(* IEC 61131-3 sources: volt/packages/volt-lsp-iec/test-corpus/pro2193/Device/Plc Logic/Application/99 Library/Function Blocks/Actuators/Cylinders, 8 files *)

(* ---- Cylinder_52Valve_InvertedFB.pou ---- *)
// Control a single output (e.g. a cylinder). Two sensors check if the cylinder is in position. The output is inverted
{attribute 'monitoring_display' := 'Output.output'}
{attribute 'symbol' := 'none'}
FUNCTION_BLOCK PUBLIC Cylinder_52Valve_InvertedFB
EXTENDS Cylinder_52ValveFB
IMPLEMENTS IActuator

%LANGUAGE ST
// Execute base cylinder fb
SUPER^();

END_FUNCTION_BLOCK

METHOD PROTECTED Alarms

%LANGUAGE ST
// Set the alarm messages (inverted)
SetSensorOutAlarm(	inputIn XOR NOT Output.Map());
SetSensorInAlarm(	inputOut XOR Output.Map());

END_METHOD

// The cylinder moves in. Returns true when cylinder is in. (Inverted!)
METHOD PUBLIC FINAL GoIn : BOOL

%LANGUAGE ST
SUPER^.GoOut();

GoIn := IsIn;

END_METHOD

// The cylinder moves out. Returns true when cylinder is out. (Inverted!)
METHOD PUBLIC FINAL GoOut : BOOL

%LANGUAGE ST
SUPER^.GoIn();

GoOut := IsOut;

END_METHOD

// Reset the output (=True, because inverted!)
METHOD Reset

%LANGUAGE ST
SUPER^.Set();

END_METHOD

// Set the output (=False, because inverted!)
METHOD Set

%LANGUAGE ST
SUPER^.Reset();

END_METHOD

// Set the output True or False (Inverted!)
METHOD SetOrReset
VAR_INPUT
	xValue	: BOOL;
END_VAR

%LANGUAGE ST
SUPER^.SetOrReset(NOT xValue);

END_METHOD

{attribute 'monitoring':='call'}
PROPERTY IsIn : BOOL

GET
VAR
END_VAR

%LANGUAGE ST
IsIn := SUPER^.IsOut;
END_GET
END_PROPERTY

{attribute 'monitoring':='call'}
PROPERTY IsOut : BOOL

GET
VAR
END_VAR

%LANGUAGE ST
IsOut := SUPER^.IsIn;
END_GET
END_PROPERTY

(* ---- Cylinder_52Valve_TimedFB.pou ---- *)
// Control a single output (e.g. a cylinder). No sensors, use timers to check cylinder position. Sensor inputs are ignored. Alarms are disabled.
{attribute 'monitoring_display' := 'Output.output'}
{attribute 'symbol' := 'none'}
FUNCTION_BLOCK PUBLIC Cylinder_52Valve_TimedFB
EXTENDS ActuatorWithManualControl_BaseFB
IMPLEMENTS IActuator
VAR_INPUT
	rTimeToGoIn				: REAL	:= 0.3;		// Time it should take for the cylinder to move in.
	rTimeToGoOut			: REAL	:= 0.3;		// Time it should take for the cylinder to move out.
END_VAR
VAR
	{attribute 'symbol' := 'read'}		Output					: ActuatorFB;

	timeGoOut				: BTON;
	timeGoIn				: BTON;

	{attribute 'symbol' := 'readwrite'}	adjustButton			: BOOL;		// Enable adjust mode for cylinder
	adjustTrigger			: TriggerFB;
	{attribute 'hide'}
	Blinker					: BLINK;	// Blinker for adjust mode
	inAdjustMode			: BOOL;		// When high the cylinder moves automatically
	SetAdjustModeTimer		: BTON;

END_VAR
VAR CONSTANT
	tAdjustFrequency		: TIME	:= T#2S;
END_VAR

%LANGUAGE ST
// Execute base fb
SUPER^();

// Instantiate the output
Output();

timeGoIn.Set(	In := NOT Output.Map(),	Pt := rTimeToGoIn);
timeGoOut.Set(	In := Output.Map(),		Pt := rTimeToGoOut);

IF adjustTrigger.Rising(CLK := adjustButton) THEN
	inAdjustMode := NOT inAdjustMode;
END_IF

inAdjustMode	S= SetAdjustModeTimer.Set(In := hardwareF1Pushed AND hardwareF2Pushed, Pt := 5);
inAdjustMode	R= plusTrigger.Q_Rising;
inAdjustMode	R= minTrigger.Q_Rising;

GlobalVars.manualControlRequested S= inAdjustMode;

Blinker(ENABLE := inAdjustMode, TIMELOW := tAdjustFrequency, TIMEHIGH := tAdjustFrequency);

END_FUNCTION_BLOCK

// The cylinder moves in. Returns true when cylinder is in.
METHOD PUBLIC FINAL GoIn : BOOL

%LANGUAGE ST
Reset();

GoIn := IsIn;

END_METHOD

// The cylinder moves out. Returns true when cylinder is out.
METHOD PUBLIC FINAL GoOut : BOOL

%LANGUAGE ST
Set();

GoOut := IsOut;

END_METHOD

METHOD PROTECTED ManualControl
VAR_INPUT
	minButtonPushed			: BOOL;		// Both the software button (on screen) and the hardware button (if attached)
	plusButtonPushed		: BOOL;		// Both the software button (on screen) and the hardware button (if attached)
END_VAR

%LANGUAGE ST
IF inAdjustMode THEN
	SetOrReset(Blinker.OUT);
ELSIF plusButtonPushed THEN
	GoOut();
ELSIF minButtonPushed THEN
	GoIn();
END_IF

END_METHOD

// Maps the actuator to the physical output
METHOD Map : BOOL

%LANGUAGE ST
Map := Output.Map();

END_METHOD

// Reset the output (=False)
METHOD Reset

%LANGUAGE ST
Output.Reset();

END_METHOD

// Set the output (=True)
METHOD Set : BOOL

%LANGUAGE ST
Output.Set();

END_METHOD

// Set the output True or False
METHOD SetOrReset
VAR_INPUT
	xValue	: BOOL;
END_VAR

%LANGUAGE ST
Output.SetOrReset(xValue);

END_METHOD

{attribute 'monitoring':='call'}
PROPERTY IsIn : BOOL

GET
VAR
END_VAR

%LANGUAGE ST
IsIn := timeGoIn.Q;
END_GET
END_PROPERTY

{attribute 'monitoring':='call'}
PROPERTY IsOut : BOOL

GET
VAR
END_VAR

%LANGUAGE ST
IsOut := timeGoOut.Q;
END_GET
END_PROPERTY

(* ---- Cylinder_52ValveFB.pou ---- *)
// Control a single output (e.g. a cylinder). Two sensors check if the cylinder is in position.
{attribute 'monitoring_display' := 'Output.output'}
{attribute 'symbol' := 'none'}
FUNCTION_BLOCK PUBLIC Cylinder_52ValveFB
EXTENDS Cylinder_BaseFB
IMPLEMENTS IActuator
VAR
	{attribute 'symbol' := 'read'}	Output					: ActuatorFB;
END_VAR

%LANGUAGE ST
// Execute base cylinder fb
SUPER^();

// Instantiate the output
Output();

END_FUNCTION_BLOCK

METHOD PROTECTED Alarms

%LANGUAGE ST
// Set the alarm messages
SetSensorOutAlarm(	inputOut XOR Output.Map());
SetSensorInAlarm(	inputIn XOR NOT Output.Map());

END_METHOD

// The cylinder moves in. Returns true when cylinder is in.
METHOD PUBLIC FINAL GoIn : BOOL

%LANGUAGE ST
Reset();

GoIn := IsIn;

END_METHOD

// The cylinder moves out. Returns true when cylinder is out.
METHOD PUBLIC FINAL GoOut : BOOL

%LANGUAGE ST
Set();

GoOut := IsOut;

END_METHOD

METHOD PROTECTED ManualControl
VAR_INPUT
	minButtonPushed			: BOOL;		// Both the software button (on screen) and the hardware button (if attached)
	plusButtonPushed		: BOOL;		// Both the software button (on screen) and the hardware button (if attached)
END_VAR

%LANGUAGE ST
IF inAdjustMode THEN
	SetOrReset(Blinker.OUT);
ELSIF plusButtonPushed THEN
	GoOut();
ELSIF minButtonPushed THEN
	GoIn();
END_IF

END_METHOD

// Maps the actuator to the physical output
METHOD Map : BOOL

%LANGUAGE ST
Map := Output.Map();

END_METHOD

// Reset the output (=False)
METHOD Reset

%LANGUAGE ST
Output.Reset();

END_METHOD

// Set the output (=True)
METHOD Set : BOOL

%LANGUAGE ST
Output.Set();

END_METHOD

// Set the output True or False
METHOD SetOrReset
VAR_INPUT
	xValue	: BOOL;
END_VAR

%LANGUAGE ST
Output.SetOrReset(xValue);

END_METHOD

(* ---- Cylinder_53Valve_InvertedFB.pou ---- *)
// Control a dual output cylinder. Two sensors check if the cylinder is in position. The outputs are inverted
{attribute 'symbol' := 'none'}
FUNCTION_BLOCK FINAL Cylinder_53Valve_InvertedFB
EXTENDS Cylinder_53ValveFB
IMPLEMENTS IActuator

%LANGUAGE ST
// Execute base cylinder fb
SUPER^();

END_FUNCTION_BLOCK

METHOD PROTECTED Alarms

%LANGUAGE ST
// Set the alarm messages (inverted)
SetSensorOutAlarm(	SetAlarm(OutputOut.Map(), OutputIn.Map(), inputIn));
SetSensorInAlarm(	SetAlarm(OutputIn.Map(), OutputOut.Map(), inputOut));

END_METHOD

// The cylinder moves in. Returns true when cylinder is in. (Inverted!)
METHOD PUBLIC GoIn : BOOL

%LANGUAGE ST
SUPER^.GoOut();

GoIn := IsIn;

END_METHOD

// The cylinder moves out. Returns true when cylinder is out. (Inverted!)
METHOD PUBLIC GoOut : BOOL

%LANGUAGE ST
SUPER^.GoIn();

GoOut := IsOut;

END_METHOD

// Set the output True or False (Inverted!)
METHOD SetOrReset
VAR_INPUT
	xValue	: BOOL;
END_VAR

%LANGUAGE ST
SUPER^.SetOrReset(NOT xValue);

END_METHOD

{attribute 'monitoring':='call'}
PROPERTY IsIn : BOOL

GET
VAR
END_VAR

%LANGUAGE ST
IsIn := SUPER^.IsOut;

END_GET
END_PROPERTY

{attribute 'monitoring':='call'}
PROPERTY IsOut : BOOL

GET
VAR
END_VAR

%LANGUAGE ST
IsOut := SUPER^.IsIn;
END_GET
END_PROPERTY

{attribute 'monitoring':='call'}
PROPERTY OnTargetPos : BOOL

GET
VAR
END_VAR

%LANGUAGE ST
OnTargetPos	:= NOT SUPER^.OnTargetPos;
END_GET
END_PROPERTY

(* ---- Cylinder_53Valve_InvertibleFB.pou ---- *)
// Control a dual output cylinder. Two sensors check if the cylinder is in position. The outputs can be inverted
{attribute 'symbol' := 'none'}
FUNCTION_BLOCK FINAL Cylinder_53Valve_InvertibleFB
EXTENDS Cylinder_53ValveFB
IMPLEMENTS IActuator
VAR_INPUT
	xInvertOutput			: BOOL;
END_VAR

%LANGUAGE ST
// Execute base cylinder fb
SUPER^();

END_FUNCTION_BLOCK

METHOD PROTECTED Alarms

%LANGUAGE ST
// Set the alarm messages (inverted)
IF xInvertOutput THEN
	SetSensorOutAlarm(	SetAlarm(OutputOut.Map(), OutputIn.Map(), inputIn));
	SetSensorInAlarm(	SetAlarm(OutputIn.Map(), OutputOut.Map(), inputOut));
ELSE
	SUPER^.Alarms();
END_IF

END_METHOD

// The cylinder moves in. Returns true when cylinder is in. (Optionally inverted!)
METHOD PUBLIC GoIn : BOOL

%LANGUAGE ST
IF xInvertOutput THEN
	SUPER^.GoOut();
ELSE
	SUPER^.GoIn();
END_IF

GoIn := IsIn;

END_METHOD

// The cylinder moves out. Returns true when cylinder is out. (Optionally inverted!)
METHOD PUBLIC GoOut : BOOL

%LANGUAGE ST
IF xInvertOutput THEN
	SUPER^.GoIn();
ELSE
	SUPER^.GoOut();
END_IF

GoOut := IsOut;

END_METHOD

// Set the output True or False
METHOD SetOrReset
VAR_INPUT
	xValue	: BOOL;
END_VAR

%LANGUAGE ST
IF xInvertOutput THEN
	SUPER^.SetOrReset(NOT xValue);
ELSE
	SUPER^.SetOrReset(xValue);
END_IF

END_METHOD

{attribute 'monitoring':='call'}
PROPERTY IsIn : BOOL

GET
VAR
END_VAR

%LANGUAGE ST
IF xInvertOutput THEN
	IsIn := SUPER^.IsOut;
ELSE
	IsIn := SUPER^.IsIn;
END_IF

END_GET
END_PROPERTY

{attribute 'monitoring':='call'}
PROPERTY IsOut : BOOL

GET
VAR
END_VAR

%LANGUAGE ST
IF xInvertOutput THEN
	IsOut := SUPER^.IsIn;
ELSE
	IsOut := SUPER^.IsOut;
END_IF

END_GET
END_PROPERTY

{attribute 'monitoring':='call'}
PROPERTY OnTargetPos : BOOL

GET
VAR
END_VAR

%LANGUAGE ST
IF xInvertOutput THEN
	OnTargetPos := NOT SUPER^.OnTargetPos;
ELSE
	OnTargetPos := SUPER^.OnTargetPos;
END_IF

END_GET
END_PROPERTY

(* ---- Cylinder_53Valve_MiddleSensorFB.pou ---- *)
// Control a dual output cylinder. Three sensors check if the cylinder is in position. Middle sensor is high when both outputs are turned off.
{attribute 'symbol' := 'none'}
FUNCTION_BLOCK FINAL Cylinder_53Valve_MiddleSensorFB
EXTENDS Cylinder_53ValveFB
VAR_INPUT
	{attribute 'symbol' := 'read'}	xSensorMiddle			: BOOL;
	errorId_SensorMiddle	: WORD;
END_VAR
VAR
	SensorMiddleAlarm		: SetErrorFB;
	{attribute 'symbol' := 'read'}		moveMiddleDuration		: REAL;		// The amount of time elapsed when cylinder moves
END_VAR

%LANGUAGE ST
// Execute base cylinder fb
SUPER^();

END_FUNCTION_BLOCK

METHOD PROTECTED Alarms

%LANGUAGE ST
// Set the extra alarm message
SUPER^.Alarms();
SetSensorMiddleAlarm(	(OutputIn.Map() = OutputOut.Map()) XOR xSensorMiddle);

END_METHOD

METHOD PROTECTED SetSensorMiddleAlarm
VAR_INPUT
	xSet	: BOOL;
END_VAR

%LANGUAGE ST
SensorMiddleAlarm(
	moduleHandler	:= moduleHandler,
	textRefId		:= textRefId,
	alarmCondition	:= alarmEnable AND xSet AND errorId_SensorMiddle <> 0,
	alarmDelay		:= alarmDelay,
	errorId			:= errorId_SensorMiddle,
	severity		:= severity,
	reaction		:= reaction,
	active			=> );

IF alarmEnable AND xSet AND errorId_SensorIn <> 0 THEN
	moveMiddleDuration	:= SensorMiddleAlarm.ElapsedTime;
END_IF

END_METHOD

{attribute 'monitoring':='call'}
PROPERTY IsIn : BOOL

GET
VAR
END_VAR

%LANGUAGE ST
IsIn := inputIn AND NOT inputOut AND NOT xSensorMiddle;
END_GET
END_PROPERTY

{attribute 'monitoring':='call'}
PROPERTY IsMiddle : BOOL

GET
VAR
END_VAR

%LANGUAGE ST
IsMiddle := NOT inputOut AND NOT inputIn AND xSensorMiddle;
END_GET
END_PROPERTY

{attribute 'monitoring':='call'}
PROPERTY IsOut : BOOL

GET
VAR
END_VAR

%LANGUAGE ST
IsOut := inputOut AND NOT inputIn AND NOT xSensorMiddle;
END_GET
END_PROPERTY

(* ---- Cylinder_53ValveFB.pou ---- *)
// Control a dual output cylinder. Two sensors check if the cylinder is in position.
{attribute 'symbol' := 'none'}
FUNCTION_BLOCK PUBLIC Cylinder_53ValveFB
EXTENDS Cylinder_BaseFB
IMPLEMENTS IActuator
VAR_INPUT
	rGiveAirToBothOutputs	: REAL := 0.2;	// When a 5/3 valve is set while both outputs are low, give air to both outputs for this time. To avoid fast moving cylinder. Default is 200MS.
	xEnableOutputs			: BOOL;			// Use like this: 'G_xEnableMainvalve OR System.On'. Resets outputs when air pressure is killed. Alarms are disables when low. Set to TRUE to disable this feature.
END_VAR
VAR
	{attribute 'symbol' := 'readwrite'}	middleButton			: BOOL;			// Enable adjust mode for cylinder
	{attribute 'symbol' := 'read'}		OutputIn				: ActuatorFB;	// Output when cylinder moves in
	{attribute 'symbol' := 'read'}		OutputOut				: ActuatorFB;	// Output when cylinder moves out

	middleTrigger			: TriggerFB;

	switchBothOutputs		: BTON;
	EnableOutputs			: BTOF;
	xStartGoInDelay			: BOOL;
	xStartGoOutDelay		: BOOL;
END_VAR

%LANGUAGE ST
// Execute base cylinder fb
SUPER^();

// Instantiate the outputs
OutputIn();
OutputOut();

// Keep xEnableOutputs high for half a second. So if air pressure drops for 0,5 sec. the outputs are reset.
IF NOT EnableOutputs.Set(In := xEnableOutputs, Pt := 0.5) THEN
	Reset();
END_IF

switchBothOutputs.Set(
	In := xStartGoInDelay OR xStartGoOutDelay,
	Pt := rGiveAirToBothOutputs);

IF switchBothOutputs.Q THEN
	SetOrReset(xStartGoOutDelay);
	xStartGoInDelay		:= FALSE;
	xStartGoOutDelay	:= FALSE;
END_IF

IF middleButton THEN
	GlobalVars.manualControlRequested := TRUE;
END_IF

END_FUNCTION_BLOCK

METHOD PROTECTED Alarms

%LANGUAGE ST
// Set the alarm messages
SetSensorOutAlarm(
	SetAlarm(
		xOutput	:= OutputOut.Map(),
		xOutInv	:= OutputIn.Map(),
		xSensor	:= inputOut));

SetSensorInAlarm(
	SetAlarm(
		xOutput	:= OutputIn.Map(),
		xOutInv	:= OutputOut.Map(),
		xSensor	:= inputIn));

END_METHOD

// Set both outputs (=True)
METHOD PUBLIC FINAL GoForceMiddle : BOOL

%LANGUAGE ST
OutputIn.Set();
OutputOut.Set();

END_METHOD

// The cylinder moves in. Returns true when cylinder is in.
METHOD PUBLIC GoIn : BOOL

%LANGUAGE ST
// Do not move cylinder if outputs are not enabled.
IF NOT EnableOutputs.Q THEN
	RETURN;
END_IF

// Both outputs are switched off, and the cylinder is not already in position
IF NOT OutputIn.Map() AND NOT OutputOut.Map() AND NOT inputIn THEN
	IF inputOut THEN		// Cylinder is on the opposite side
		OutputOut.Set();		// Send cylinder to opposite direction
		OutputIn.Reset();
		xStartGoInDelay	:= TRUE;
	ELSE					// Cylinder is in between sensors
		GoForceMiddle();	// Give air to both sides of the cylinder
		xStartGoInDelay	:= TRUE;
	END_IF
ELSIF NOT xStartGoInDelay THEN
	OutputOut.Reset();
	OutputIn.Set();

	GoIn := IsIn;
END_IF

END_METHOD

// Reset both outputs. The 5/3 valve goes to middle position.
METHOD PUBLIC GoMiddle

%LANGUAGE ST
Reset();
END_METHOD

// The cylinder moves out. Returns true when cylinder is out.
METHOD PUBLIC GoOut : BOOL

%LANGUAGE ST
// Do not move cylinder if outputs are not enabled.
IF NOT EnableOutputs.Q THEN
	RETURN;
END_IF

// Both outputs are switched off, and the cylinder is not already in position
IF NOT OutputIn.Map() AND NOT OutputOut.Map() AND NOT inputOut THEN
	IF inputIn THEN		// Cylinder is on the opposite side
		OutputOut.Reset();
		OutputIn.Set();		// Send cylinder to opposite direction
		xStartGoOutDelay	:= TRUE;
	ELSE					// Cylinder is in between sensors
		GoForceMiddle();	// Give air to both sides of the cylinder
		xStartGoOutDelay	:= TRUE;
	END_IF
ELSIF NOT xStartGoOutDelay THEN
	OutputOut.Set();
	OutputIn.Reset();

	GoOut := IsOut;
END_IF

END_METHOD

METHOD PROTECTED ManualControl
VAR_INPUT
	minButtonPushed			: BOOL;		// Both the software button (on screen) and the hardware button (if attached)
	plusButtonPushed		: BOOL;		// Both the software button (on screen) and the hardware button (if attached)
END_VAR

%LANGUAGE ST
IF inAdjustMode THEN
	SetOrReset(Blinker.OUT);
ELSIF plusButtonPushed THEN
	IF OutputOut.Map() THEN
		GoMiddle();
	ELSE
		GoOut();
	END_IF
ELSIF minButtonPushed THEN
	IF OutputIn.Map() THEN
		GoMiddle();
	ELSE
		GoIn();
	END_IF
ELSIF middleTrigger.Rising(CLK := middleButton) THEN
	GoMiddle();
END_IF

END_METHOD

{attribute 'hide'}
METHOD Map : BOOL

%LANGUAGE ST
ThrowException('Use other mapping methods instead');

END_METHOD

// Maps the output when cylinder moves Out to the physical output
METHOD MapIn : BOOL

%LANGUAGE ST
MapIn := OutputIn.Map();

END_METHOD

// Maps the output when cylinder moves Out to the physical output
METHOD MapOut : BOOL

%LANGUAGE ST
MapOut := OutputOut.Map();

END_METHOD

// Reset the outputs (=False)
METHOD Reset

%LANGUAGE ST
OutputIn.Reset();
OutputOut.Reset();

END_METHOD

// Set the outputs (=True)
METHOD Set : BOOL

%LANGUAGE ST
GoOut();

END_METHOD

METHOD PRIVATE SetAlarm : BOOL
VAR_INPUT
	xOutput		: BOOL;		// The output
	xOutInv		: BOOL;		// The output that moves the cylinder the other way.
	xSensor		: BOOL;		// The sensor on the cylinder.
END_VAR

%LANGUAGE FBD
%NETWORK
ASSIGN(AND(AND(xOutput, INVERT(xOutInv), INVERT(xSensor)) OR AND(xOutInv, INVERT(xOutput), xSensor) OR AND(xOutput, xOutInv, xSensor), EnableOutputs.Q), Q => SetAlarm);
END_METHOD

// Set the output True or False
METHOD SetOrReset
VAR_INPUT
	xValue	: BOOL;
END_VAR

%LANGUAGE ST
// Do not move cylinder if outputs are not enabled.
IF NOT EnableOutputs.Q THEN
	RETURN;
END_IF

// Timer expired, so both outputs are high. Just switch to desired output.
IF switchBothOutputs.Q THEN
	OutputOut.SetOrReset(xValue);
	OutputIn.SetOrReset(NOT xValue);
// Both outputs are switched off. Give air to both sides of the valve. Start timer.
ELSIF NOT OutputIn.Map() AND NOT OutputOut.Map() THEN
	GoForceMiddle();
	xStartGoInDelay		:= NOT xValue;	// Choose direction to move to when timer expires.
	xStartGoOutDelay	:= xValue;
// Normal operation
ELSIF NOT xStartGoInDelay AND NOT xStartGoOutDelay THEN
	OutputOut.SetOrReset(xValue);
	OutputIn.SetOrReset(NOT xValue);
END_IF

END_METHOD

// Set both the outputs of the valve immediately
METHOD SetOrResetBothOutputs : BOOL
VAR_INPUT
	xOutput2	: BOOL;		// Output when cylinder moves out
	xOutput1	: BOOL;		// Output when cylinder moves in
END_VAR

%LANGUAGE ST
OutputOut.SetOrReset(xOutput2);
OutputIn.SetOrReset(xOutput1);

END_METHOD

{attribute 'monitoring':='call'}
PROPERTY OnTargetPos : BOOL

GET
VAR
END_VAR

%LANGUAGE ST
OnTargetPos	:= NOT xStartGoInDelay AND NOT xStartGoOutDelay AND EnableOutputs.Q AND
			(OutputOut.Map() AND NOT OutputIn.Map() AND IsOut) XOR (OutputIn.Map() AND NOT OutputOut.Map() AND IsIn);

END_GET
END_PROPERTY

(* ---- Cylinder_BaseFB.pou ---- *)
// Abstract Base fb for cylinders. Has general stuff for all cylinder types.
{attribute 'symbol' := 'none'}
FUNCTION_BLOCK PUBLIC ABSTRACT Cylinder_BaseFB
EXTENDS ActuatorWithManualControlAndAlarm_BaseFB
VAR_INPUT
	{attribute 'symbol' := 'read'}		inputOut				: BOOL;
	{attribute 'symbol' := 'read'}		inputIn					: BOOL;
	errorId_SensorOut		: WORD;		// Set to ZERO if OUT sensor is not on the cylinder, this will prevent incorrect alarm messages.
	errorId_SensorIn		: WORD;		// Set to ZERO if IN sensor is not on the cylinder, this will prevent incorrect alarm messages.
END_VAR
VAR
	SensorOutAlarm			: SetErrorFB;
	SensorInAlarm			: SetErrorFB;
	{attribute 'symbol' := 'read'}		moveInDuration			: REAL;		// The amount of time elapsed when cylinder moves out
	{attribute 'symbol' := 'read'}		moveOutDuration			: REAL;		// The amount of time elapsed when cylinder moves in

	MeasureMaxTimeIn		: StopwatchFB;
	MeasureMaxTimeOut		: StopwatchFB;

	{attribute 'symbol' := 'readwrite'}	adjustButton			: BOOL;		// Enable adjust mode for cylinder
	adjustTrigger			: TriggerFB;
	{attribute 'hide'}
	Blinker					: BLINK;	// Blinker for adjust mode
	inAdjustMode			: BOOL;		// When high the cylinder moves automatically
	SetAdjustModeTimer		: BTON;
END_VAR
VAR CONSTANT
	tAdjustFrequency		: TIME	:= T#2S;
END_VAR

%LANGUAGE ST
SUPER^();

IF adjustTrigger.Rising(CLK := adjustButton) THEN
	inAdjustMode := NOT inAdjustMode;
END_IF

inAdjustMode	S= SetAdjustModeTimer.Set(In := hardwareF1Pushed AND hardwareF2Pushed, Pt := 5);
inAdjustMode	R= plusTrigger.Q_Rising;
inAdjustMode	R= minTrigger.Q_Rising;

GlobalVars.manualControlRequested S= inAdjustMode;

Blinker(ENABLE := inAdjustMode, TIMELOW := tAdjustFrequency, TIMEHIGH := tAdjustFrequency);

END_FUNCTION_BLOCK

METHOD PUBLIC SetMonitoring
VAR_INPUT
	itfAddLog		: EdgePcLogging.IAddLog;
	plcDataTypeIn	: PlcDataType;
	plcDataTypeOut	: PlcDataType;
END_VAR

%LANGUAGE ST
IF errorId_SensorOut <> 0 THEN
	MeasureMaxTimeIn.SetMonitoring(		itfAddLog, plcDataTypeIn);
END_IF

IF errorId_SensorIn <> 0 THEN
	MeasureMaxTimeOut.SetMonitoring(	itfAddLog, plcDataTypeOut);
END_IF

END_METHOD

METHOD PROTECTED SetSensorInAlarm
VAR_INPUT
	xSet	: BOOL;
END_VAR

%LANGUAGE ST
SensorInAlarm(
	moduleHandler	:= moduleHandler,
	textRefId		:= textRefId,
	alarmCondition	:= alarmEnable AND xSet AND errorId_SensorIn <> 0,
	alarmDelay		:= alarmDelay,
	errorId			:= errorId_SensorIn,
	severity		:= severity,
	reaction		:= reaction,
	active			=> );

IF alarmEnable AND xSet AND NOT inputIn AND errorId_SensorIn <> 0 THEN
	moveInDuration	:= SensorInAlarm.ElapsedTime;
END_IF

MeasureMaxTimeIn.Monitor(
	in				:= xSet AND NOT inputIn AND errorId_SensorIn <> 0);

END_METHOD

METHOD PROTECTED SetSensorOutAlarm
VAR_INPUT
	xSet	: BOOL;
END_VAR

%LANGUAGE ST
SensorOutAlarm(
	moduleHandler	:= moduleHandler,
	textRefId		:= textRefId,
	alarmCondition	:= alarmEnable AND xSet AND errorId_SensorOut <> 0,
	alarmDelay		:= alarmDelay,
	errorId			:= errorId_SensorOut,
	severity		:= severity,
	reaction		:= reaction,
	active			=> );

IF alarmEnable AND xSet AND NOT inputOut AND errorId_SensorIn <> 0 THEN
	moveOutDuration	:= SensorOutAlarm.ElapsedTime;
END_IF

MeasureMaxTimeOut.Monitor(
	in				:= xSet AND NOT inputOut AND errorId_SensorOut <> 0);

END_METHOD

{attribute 'monitoring':='call'}
PROPERTY IsIn : BOOL

GET
VAR
END_VAR

%LANGUAGE ST
IsIn := inputIn AND NOT inputOut;
END_GET
END_PROPERTY

{attribute 'monitoring':='call'}
PROPERTY IsOut : BOOL

GET
VAR
END_VAR

%LANGUAGE ST
IsOut := inputOut AND NOT inputIn;
END_GET
END_PROPERTY
